FUNCTION_BLOCK UNIT_StateIds (* OPC UA IDs of the unit commands and state *)
  (* Standard: 61499-2 *)
  (* Version 0.1, 2026-09-28, Project contributors, AAU Smart Production Lab *)
  PACKAGE unitlib;
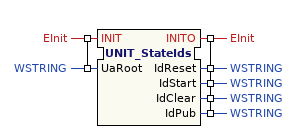
  EVENT_INPUT
    INIT : EInit WITH UaRoot;
  END_EVENT
  EVENT_OUTPUT
    INITO : EInit WITH IdReset, IdStart, IdClear, IdPub;
  END_EVENT
  VAR_INPUT
    UaRoot : WSTRING;
  END_VAR
  VAR_OUTPUT
    IdReset : WSTRING;
    IdStart : WSTRING;
    IdClear : WSTRING;
    IdPub : WSTRING;
  END_VAR
  EC_STATES
    INIT : INIT -> INITO;
  END_STATES
  ALGORITHM INIT IN ST:
IdReset := CONCAT(CONCAT("opc_ua[CREATE_METHOD;", CONCAT(UaRoot, "/Unit/")), "Reset]");
IdStart := CONCAT(CONCAT("opc_ua[CREATE_METHOD;", CONCAT(UaRoot, "/Unit/")), "Start]");
IdClear := CONCAT(CONCAT("opc_ua[CREATE_METHOD;", CONCAT(UaRoot, "/Unit/")), "Clear]");
IdPub := CONCAT(CONCAT("opc_ua[WRITE;", CONCAT(UaRoot, "/Unit/")), "State]");
  END_ALGORITHM
END_FUNCTION_BLOCK
